// TIA Portal V20 export
DATA_BLOCK "ET500SP_505"   // DB235
// stored: MemoryReserve 100
   VAR
      "SP505.00 UNWINDER DANCER ELECTRO-PNEUMATIC REGULATOR" : LReal;
      SPARE1 : LReal;
      SPARE2 : LReal;
      SPARE3 : LReal;
   END_VAR
BEGIN
END_DATA_BLOCK
